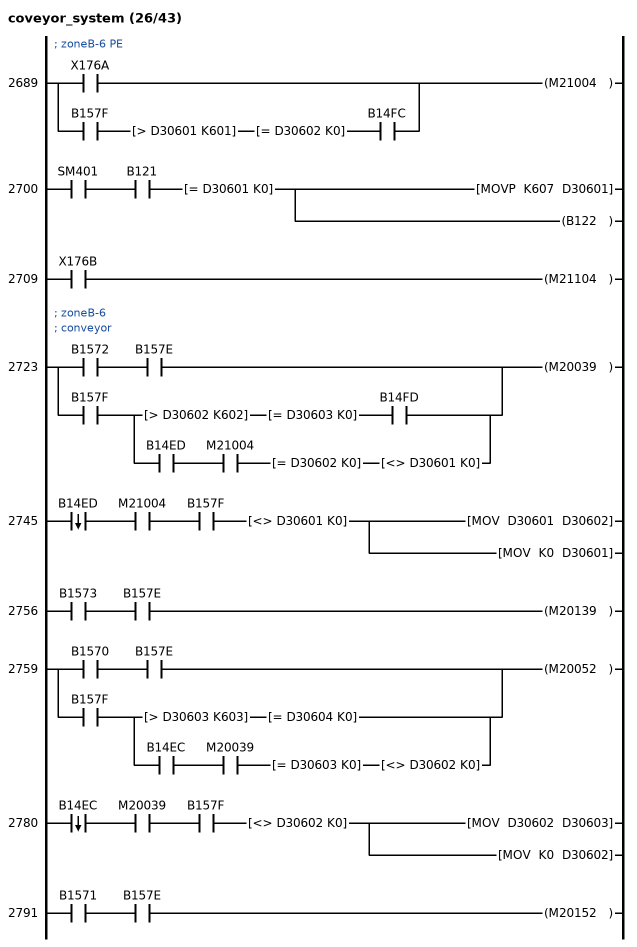
[picture p192: ladder of coveyor_system, rungs at steps 2689 to 2791]
; zoneB-6 PE
2689  LD      X176A
      LD      B157F
      AND>    D30601 K601
      AND=    D30602 K0
      AND     B14FC
      ORB
      OUT     M21004
2700  LD      SM401
      AND     B121
      AND=    D30601 K0
      MOVP    K607 D30601
      OUT     B122
2709  LD      X176B
      OUT     M21104
; zoneB-6
; conveyor
2723  LD      B1572
      AND     B157E
      LD      B157F
      LD>     D30602 K602
      AND=    D30603 K0
      AND     B14FD
      LD      B14ED
      AND     M21004
      AND=    D30602 K0
      AND<>   D30601 K0
      ORB
      ANB
      ORB
      OUT     M20039
2745  LDF     B14ED
      AND     M21004
      AND     B157F
      AND<>   D30601 K0
      MOV     D30601 D30602
      MOV     K0 D30601
2756  LD      B1573
      AND     B157E
      OUT     M20139
2759  LD      B1570
      AND     B157E
      LD      B157F
      LD>     D30603 K603
      AND=    D30604 K0
      LD      B14EC
      AND     M20039
      AND=    D30603 K0
      AND<>   D30602 K0
      ORB
      ANB
      ORB
      OUT     M20052
2780  LDF     B14EC
      AND     M20039
      AND     B157F
      AND<>   D30602 K0
      MOV     D30602 D30603
      MOV     K0 D30602
2791  LD      B1571
      AND     B157E
      OUT     M20152
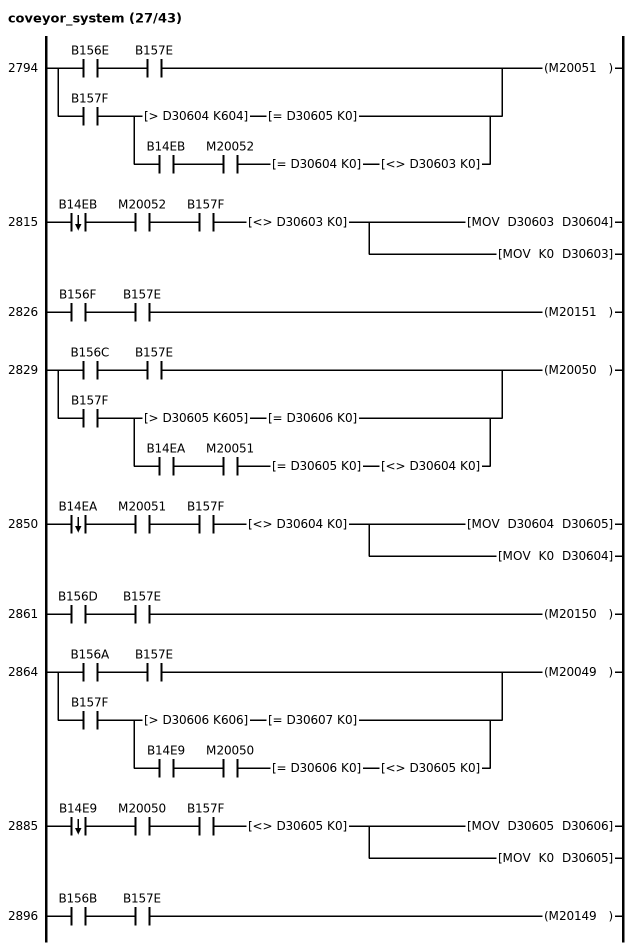
2794  LD      B156E
      AND     B157E
      LD      B157F
      LD>     D30604 K604
      AND=    D30605 K0
      LD      B14EB
      AND     M20052
      AND=    D30604 K0
      AND<>   D30603 K0
      ORB
      ANB
      ORB
      OUT     M20051
2815  LDF     B14EB
      AND     M20052
      AND     B157F
      AND<>   D30603 K0
      MOV     D30603 D30604
      MOV     K0 D30603
2826  LD      B156F
      AND     B157E
      OUT     M20151
2829  LD      B156C
      AND     B157E
      LD      B157F
      LD>     D30605 K605
      AND=    D30606 K0
      LD      B14EA
      AND     M20051
      AND=    D30605 K0
      AND<>   D30604 K0
      ORB
      ANB
      ORB
      OUT     M20050
2850  LDF     B14EA
      AND     M20051
      AND     B157F
      AND<>   D30604 K0
      MOV     D30604 D30605
      MOV     K0 D30604
2861  LD      B156D
      AND     B157E
      OUT     M20150
2864  LD      B156A
      AND     B157E
      LD      B157F
      LD>     D30606 K606
      AND=    D30607 K0
      LD      B14E9
      AND     M20050
      AND=    D30606 K0
      AND<>   D30605 K0
      ORB
      ANB
      ORB
      OUT     M20049
2885  LDF     B14E9
      AND     M20050
      AND     B157F
      AND<>   D30605 K0
      MOV     D30605 D30606
      MOV     K0 D30605
2896  LD      B156B
      AND     B157E
      OUT     M20149
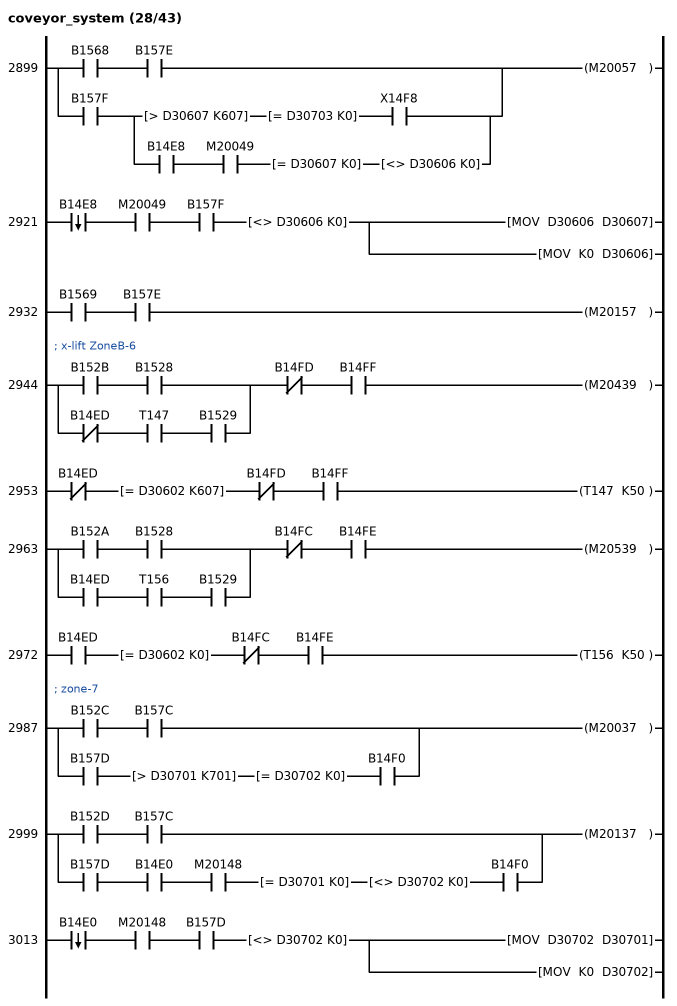
2899  LD      B1568
      AND     B157E
      LD      B157F
      LD>     D30607 K607
      AND=    D30703 K0
      AND     X14F8
      LD      B14E8
      AND     M20049
      AND=    D30607 K0
      AND<>   D30606 K0
      ORB
      ANB
      ORB
      OUT     M20057
2921  LDF     B14E8
      AND     M20049
      AND     B157F
      AND<>   D30606 K0
      MOV     D30606 D30607
      MOV     K0 D30606
2932  LD      B1569
      AND     B157E
      OUT     M20157
; x-lift ZoneB-6
2944  LD      B152B
      AND     B1528
      LDI     B14ED
      AND     T147
      AND     B1529
      ORB
      ANI     B14FD
      AND     B14FF
      OUT     M20439
2953  LDI     B14ED
      AND=    D30602 K607
      ANI     B14FD
      AND     B14FF
      OUT     T147 K50
2963  LD      B152A
      AND     B1528
      LD      B14ED
      AND     T156
      AND     B1529
      ORB
      ANI     B14FC
      AND     B14FE
      OUT     M20539
2972  LD      B14ED
      AND=    D30602 K0
      ANI     B14FC
      AND     B14FE
      OUT     T156 K50
; zone-7
2987  LD      B152C
      AND     B157C
      LD      B157D
      AND>    D30701 K701
      AND=    D30702 K0
      AND     B14F0
      ORB
      OUT     M20037
2999  LD      B152D
      AND     B157C
      LD      B157D
      AND     B14E0
      AND     M20148
      AND=    D30701 K0
      AND<>   D30702 K0
      AND     B14F0
      ORB
      OUT     M20137
3013  LDF     B14E0
      AND     M20148
      AND     B157D
      AND<>   D30702 K0
      MOV     D30702 D30701
      MOV     K0 D30702
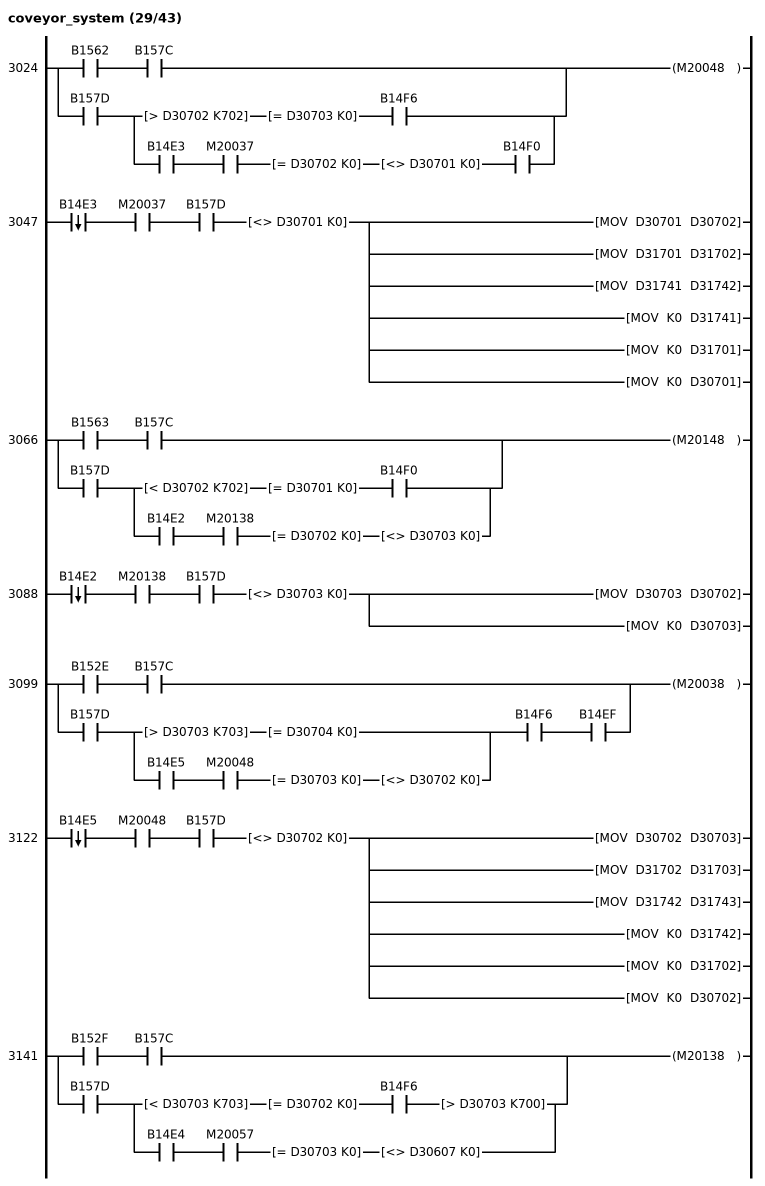
3024  LD      B1562
      AND     B157C
      LD      B157D
      LD>     D30702 K702
      AND=    D30703 K0
      AND     B14F6
      LD      B14E3
      AND     M20037
      AND=    D30702 K0
      AND<>   D30701 K0
      AND     B14F0
      ORB
      ANB
      ORB
      OUT     M20048
3047  LDF     B14E3
      AND     M20037
      AND     B157D
      AND<>   D30701 K0
      MOV     D30701 D30702
      MOV     D31701 D31702
      MOV     D31741 D31742
      MOV     K0 D31741
      MOV     K0 D31701
      MOV     K0 D30701
3066  LD      B1563
      AND     B157C
      LD      B157D
      LD<     D30702 K702
      AND=    D30701 K0
      AND     B14F0
      LD      B14E2
      AND     M20138
      AND=    D30702 K0
      AND<>   D30703 K0
      ORB
      ANB
      ORB
      OUT     M20148
3088  LDF     B14E2
      AND     M20138
      AND     B157D
      AND<>   D30703 K0
      MOV     D30703 D30702
      MOV     K0 D30703
3099  LD      B152E
      AND     B157C
      LD      B157D
      LD>     D30703 K703
      AND=    D30704 K0
      LD      B14E5
      AND     M20048
      AND=    D30703 K0
      AND<>   D30702 K0
      ORB
      ANB
      AND     B14F6
      AND     B14EF
      ORB
      OUT     M20038
3122  LDF     B14E5
      AND     M20048
      AND     B157D
      AND<>   D30702 K0
      MOV     D30702 D30703
      MOV     D31702 D31703
      MOV     D31742 D31743
      MOV     K0 D31742
      MOV     K0 D31702
      MOV     K0 D30702
3141  LD      B152F
      AND     B157C
      LD      B157D
      LD<     D30703 K703
      AND=    D30702 K0
      AND     B14F6
      AND>    D30703 K700
      LD      B14E4
      AND     M20057
      AND=    D30703 K0
      AND<>   D30607 K0
      ORB
      ANB
      ORB
      OUT     M20138
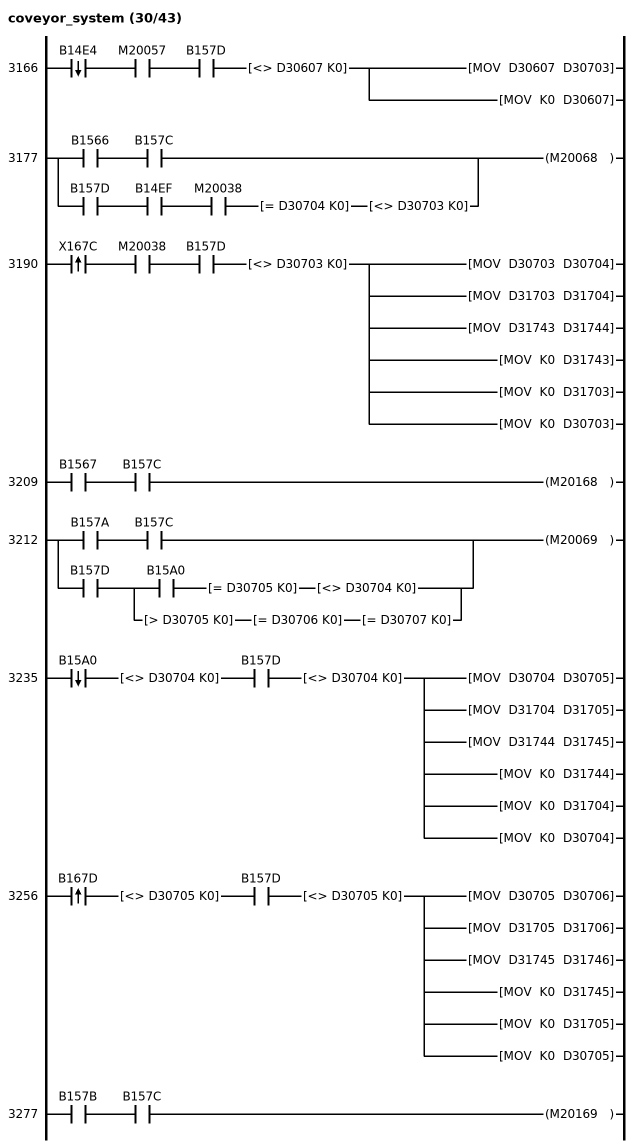
3166  LDF     B14E4
      AND     M20057
      AND     B157D
      AND<>   D30607 K0
      MOV     D30607 D30703
      MOV     K0 D30607
3177  LD      B1566
      AND     B157C
      LD      B157D
      AND     B14EF
      AND     M20038
      AND=    D30704 K0
      AND<>   D30703 K0
      ORB
      OUT     M20068
3190  LDP     X167C
      AND     M20038
      AND     B157D
      AND<>   D30703 K0
      MOV     D30703 D30704
      MOV     D31703 D31704
      MOV     D31743 D31744
      MOV     K0 D31743
      MOV     K0 D31703
      MOV     K0 D30703
3209  LD      B1567
      AND     B157C
      OUT     M20168
3212  LD      B157A
      AND     B157C
      LD      B157D
      LD      B15A0
      AND=    D30705 K0
      AND<>   D30704 K0
      LD>     D30705 K0
      AND=    D30706 K0
      AND=    D30707 K0
      ORB
      ANB
      ORB
      OUT     M20069
3235  LDF     B15A0
      AND<>   D30704 K0
      AND     B157D
      AND<>   D30704 K0
      MOV     D30704 D30705
      MOV     D31704 D31705
      MOV     D31744 D31745
      MOV     K0 D31744
      MOV     K0 D31704
      MOV     K0 D30704
3256  LDP     B167D
      AND<>   D30705 K0
      AND     B157D
      AND<>   D30705 K0
      MOV     D30705 D30706
      MOV     D31705 D31706
      MOV     D31745 D31746
      MOV     K0 D31745
      MOV     K0 D31705
      MOV     K0 D30705
3277  LD      B157B
      AND     B157C
      OUT     M20169
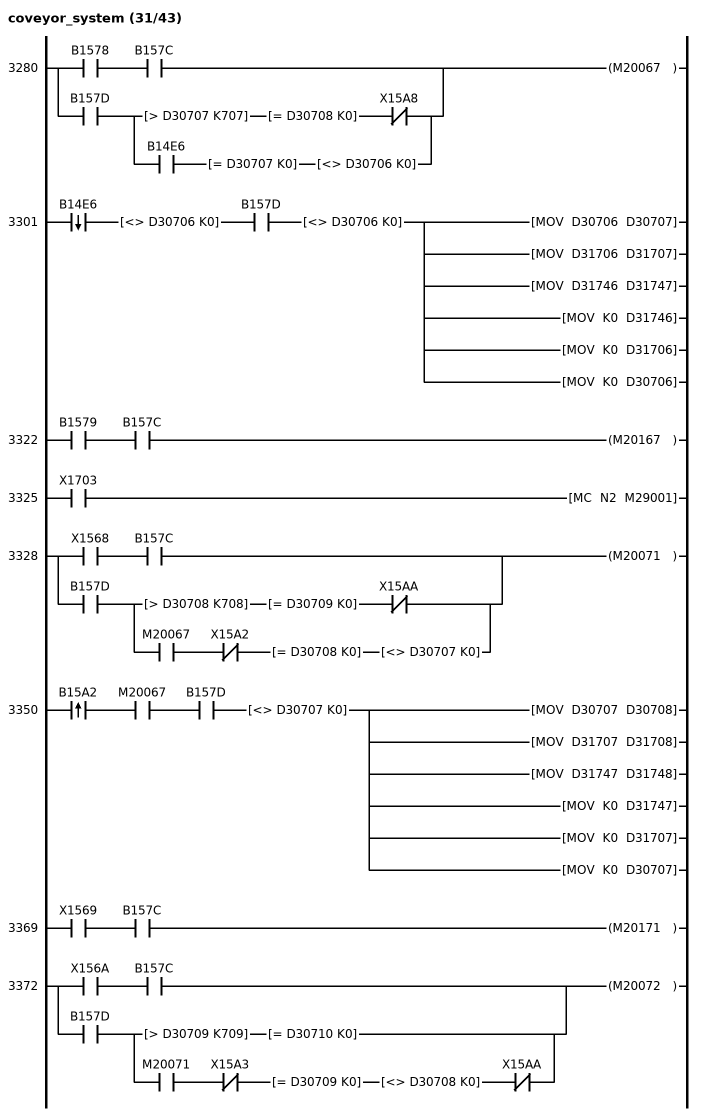
3280  LD      B1578
      AND     B157C
      LD      B157D
      LD>     D30707 K707
      AND=    D30708 K0
      ANI     X15A8
      LD      B14E6
      AND=    D30707 K0
      AND<>   D30706 K0
      ORB
      ANB
      ORB
      OUT     M20067
3301  LDF     B14E6
      AND<>   D30706 K0
      AND     B157D
      AND<>   D30706 K0
      MOV     D30706 D30707
      MOV     D31706 D31707
      MOV     D31746 D31747
      MOV     K0 D31746
      MOV     K0 D31706
      MOV     K0 D30706
3322  LD      B1579
      AND     B157C
      OUT     M20167
3325  LD      X1703
      MC      N2 M29001
3328  LD      X1568
      AND     B157C
      LD      B157D
      LD>     D30708 K708
      AND=    D30709 K0
      ANI     X15AA
      LD      M20067
      ANI     X15A2
      AND=    D30708 K0
      AND<>   D30707 K0
      ORB
      ANB
      ORB
      OUT     M20071
3350  LDP     B15A2
      AND     M20067
      AND     B157D
      AND<>   D30707 K0
      MOV     D30707 D30708
      MOV     D31707 D31708
      MOV     D31747 D31748
      MOV     K0 D31747
      MOV     K0 D31707
      MOV     K0 D30707
3369  LD      X1569
      AND     B157C
      OUT     M20171
3372  LD      X156A
      AND     B157C
      LD      B157D
      LD>     D30709 K709
      AND=    D30710 K0
      LD      M20071
      ANI     X15A3
      AND=    D30709 K0
      AND<>   D30708 K0
      ANI     X15AA
      ORB
      ANB
      ORB
      OUT     M20072
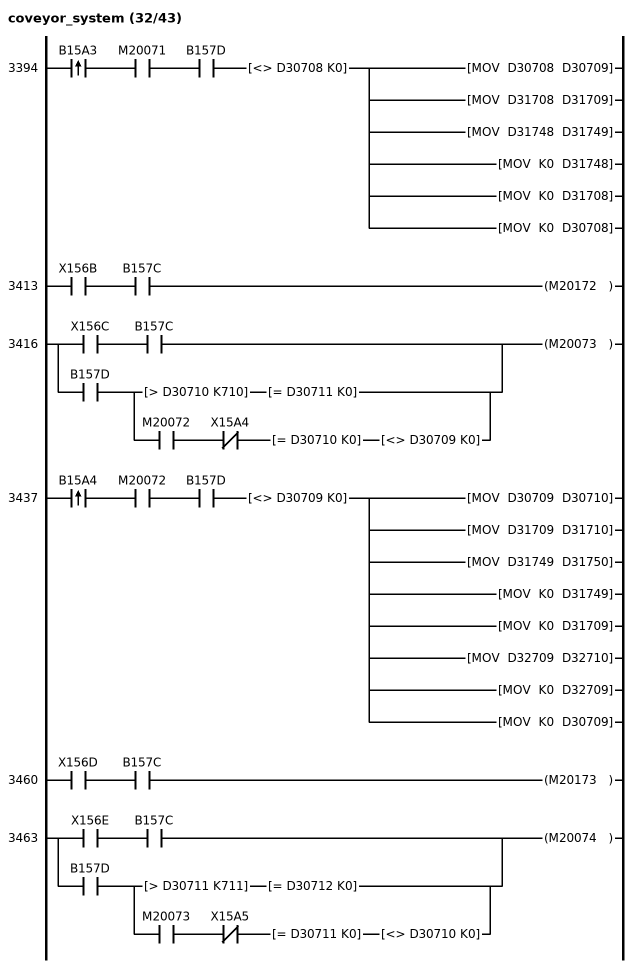
3394  LDP     B15A3
      AND     M20071
      AND     B157D
      AND<>   D30708 K0
      MOV     D30708 D30709
      MOV     D31708 D31709
      MOV     D31748 D31749
      MOV     K0 D31748
      MOV     K0 D31708
      MOV     K0 D30708
3413  LD      X156B
      AND     B157C
      OUT     M20172
3416  LD      X156C
      AND     B157C
      LD      B157D
      LD>     D30710 K710
      AND=    D30711 K0
      LD      M20072
      ANI     X15A4
      AND=    D30710 K0
      AND<>   D30709 K0
      ORB
      ANB
      ORB
      OUT     M20073
3437  LDP     B15A4
      AND     M20072
      AND     B157D
      AND<>   D30709 K0
      MOV     D30709 D30710
      MOV     D31709 D31710
      MOV     D31749 D31750
      MOV     K0 D31749
      MOV     K0 D31709
      MOV     D32709 D32710
      MOV     K0 D32709
      MOV     K0 D30709
3460  LD      X156D
      AND     B157C
      OUT     M20173
3463  LD      X156E
      AND     B157C
      LD      B157D
      LD>     D30711 K711
      AND=    D30712 K0
      LD      M20073
      ANI     X15A5
      AND=    D30711 K0
      AND<>   D30710 K0
      ORB
      ANB
      ORB
      OUT     M20074
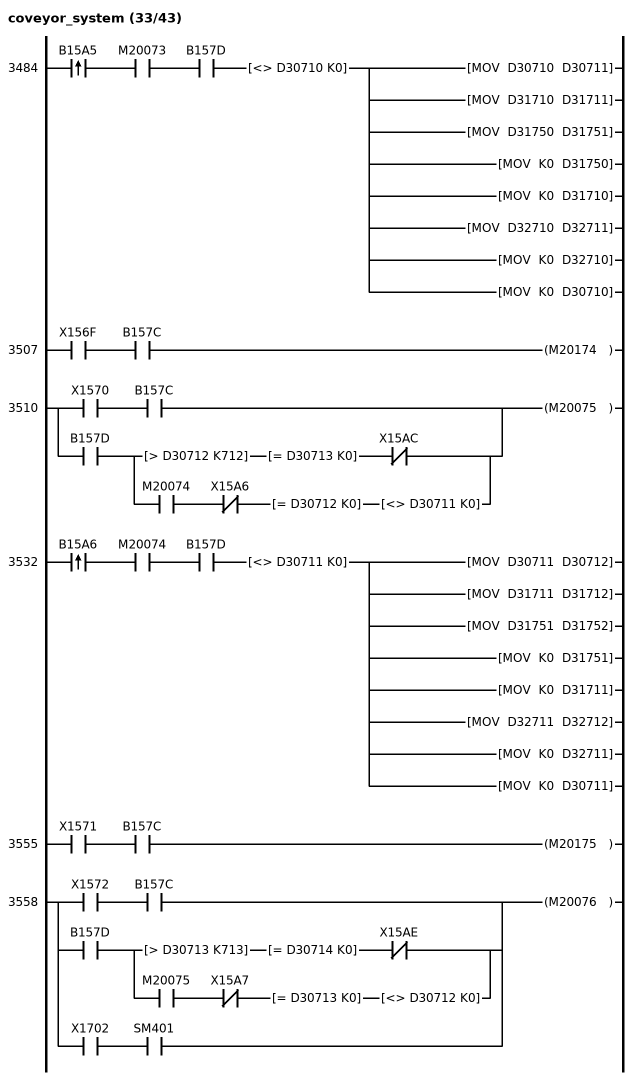
3484  LDP     B15A5
      AND     M20073
      AND     B157D
      AND<>   D30710 K0
      MOV     D30710 D30711
      MOV     D31710 D31711
      MOV     D31750 D31751
      MOV     K0 D31750
      MOV     K0 D31710
      MOV     D32710 D32711
      MOV     K0 D32710
      MOV     K0 D30710
3507  LD      X156F
      AND     B157C
      OUT     M20174
3510  LD      X1570
      AND     B157C
      LD      B157D
      LD>     D30712 K712
      AND=    D30713 K0
      ANI     X15AC
      LD      M20074
      ANI     X15A6
      AND=    D30712 K0
      AND<>   D30711 K0
      ORB
      ANB
      ORB
      OUT     M20075
3532  LDP     B15A6
      AND     M20074
      AND     B157D
      AND<>   D30711 K0
      MOV     D30711 D30712
      MOV     D31711 D31712
      MOV     D31751 D31752
      MOV     K0 D31751
      MOV     K0 D31711
      MOV     D32711 D32712
      MOV     K0 D32711
      MOV     K0 D30711
3555  LD      X1571
      AND     B157C
      OUT     M20175
3558  LD      X1572
      AND     B157C
      LD      B157D
      LD>     D30713 K713
      AND=    D30714 K0
      ANI     X15AE
      LD      M20075
      ANI     X15A7
      AND=    D30713 K0
      AND<>   D30712 K0
      ORB
      ANB
      ORB
      LD      X1702
      AND     SM401
      ORB
      OUT     M20076
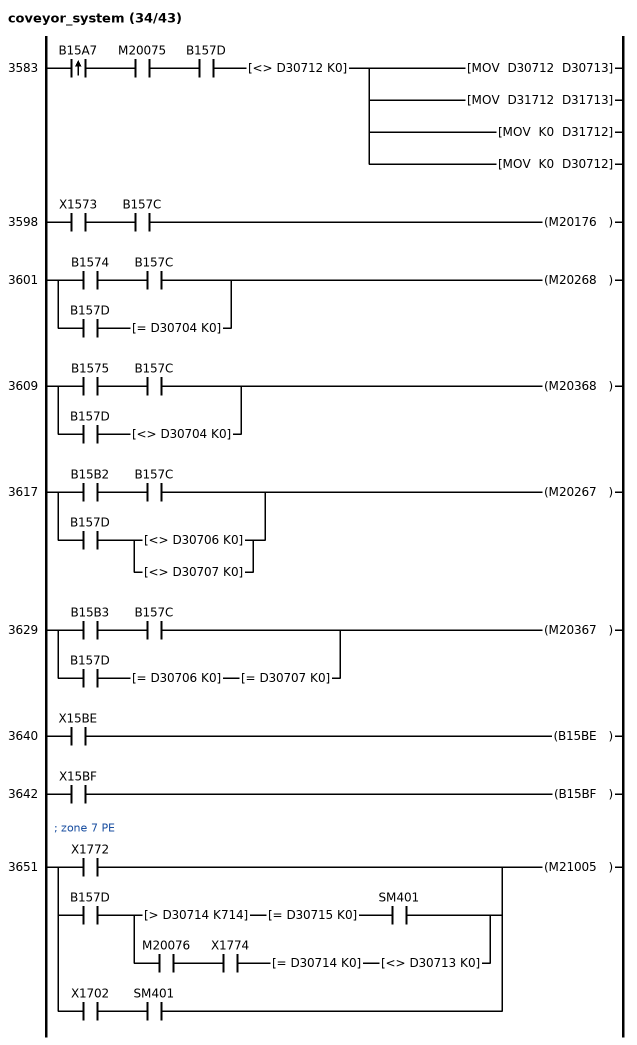
3583  LDP     B15A7
      AND     M20075
      AND     B157D
      AND<>   D30712 K0
      MOV     D30712 D30713
      MOV     D31712 D31713
      MOV     K0 D31712
      MOV     K0 D30712
3598  LD      X1573
      AND     B157C
      OUT     M20176
3601  LD      B1574
      AND     B157C
      LD      B157D
      AND=    D30704 K0
      ORB
      OUT     M20268
3609  LD      B1575
      AND     B157C
      LD      B157D
      AND<>   D30704 K0
      ORB
      OUT     M20368
3617  LD      B15B2
      AND     B157C
      LD      B157D
      LD<>    D30706 K0
      OR<>    D30707 K0
      ANB
      ORB
      OUT     M20267
3629  LD      B15B3
      AND     B157C
      LD      B157D
      AND=    D30706 K0
      AND=    D30707 K0
      ORB
      OUT     M20367
3640  LD      X15BE
      OUT     B15BE
3642  LD      X15BF
      OUT     B15BF
; zone 7 PE
3651  LD      X1772
      LD      B157D
      LD>     D30714 K714
      AND=    D30715 K0
      AND     SM401
      LD      M20076
      AND     X1774
      AND=    D30714 K0
      AND<>   D30713 K0
      ORB
      ANB
      ORB
      LD      X1702
      AND     SM401
      ORB
      OUT     M21005
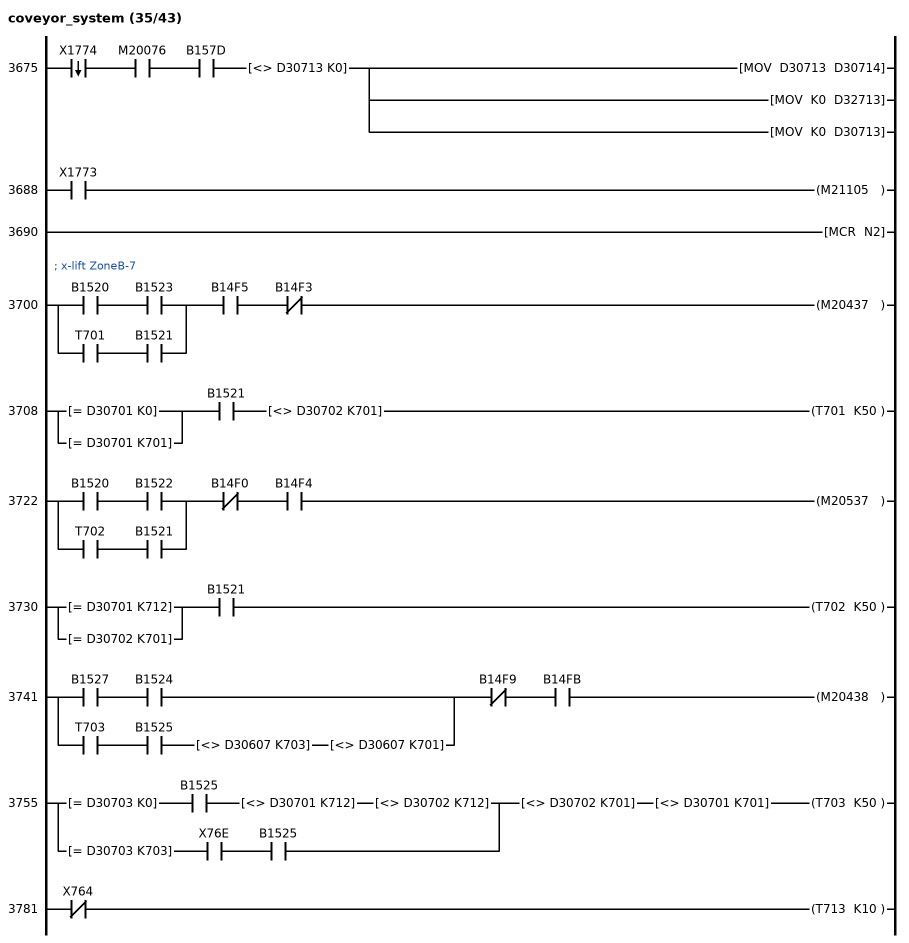
3675  LDF     X1774
      AND     M20076
      AND     B157D
      AND<>   D30713 K0
      MOV     D30713 D30714
      MOV     K0 D32713
      MOV     K0 D30713
3688  LD      X1773
      OUT     M21105
3690  MCR     N2
; x-lift ZoneB-7
3700  LD      B1520
      AND     B1523
      LD      T701
      AND     B1521
      ORB
      AND     B14F5
      ANI     B14F3
      OUT     M20437
3708  LD=     D30701 K0
      OR=     D30701 K701
      AND     B1521
      AND<>   D30702 K701
      OUT     T701 K50
3722  LD      B1520
      AND     B1522
      LD      T702
      AND     B1521
      ORB
      ANI     B14F0
      AND     B14F4
      OUT     M20537
3730  LD=     D30701 K712
      OR=     D30702 K701
      AND     B1521
      OUT     T702 K50
3741  LD      B1527
      AND     B1524
      LD      T703
      AND     B1525
      AND<>   D30607 K703
      AND<>   D30607 K701
      ORB
      ANI     B14F9
      AND     B14FB
      OUT     M20438
3755  LD=     D30703 K0
      AND     B1525
      AND<>   D30701 K712
      AND<>   D30702 K712
      LD=     D30703 K703
      AND     X76E
      AND     B1525
      ORB
      AND<>   D30702 K701
      AND<>   D30701 K701
      OUT     T703 K50
3781  LDI     X764
      OUT     T713 K10
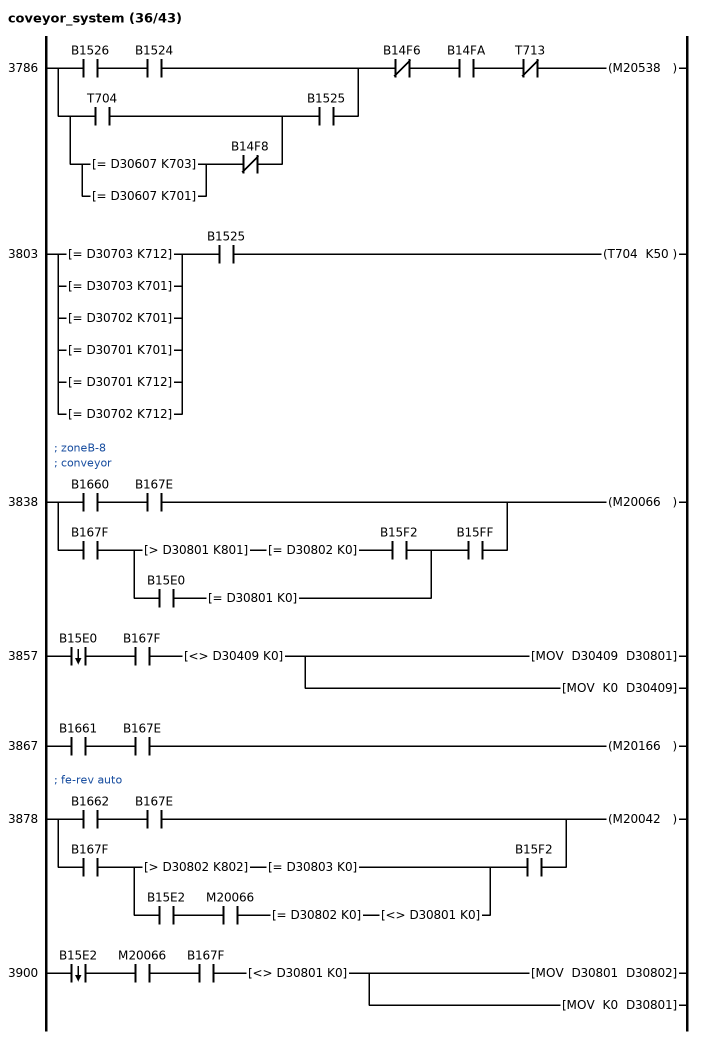
3786  LD      B1526
      AND     B1524
      LD      T704
      LD=     D30607 K703
      OR=     D30607 K701
      ANI     B14F8
      ORB
      AND     B1525
      ORB
      ANI     B14F6
      AND     B14FA
      ANI     T713
      OUT     M20538
3803  LD=     D30703 K712
      OR=     D30703 K701
      OR=     D30702 K701
      OR=     D30701 K701
      OR=     D30701 K712
      OR=     D30702 K712
      AND     B1525
      OUT     T704 K50
; zoneB-8
; conveyor
3838  LD      B1660
      AND     B167E
      LD      B167F
      LD>     D30801 K801
      AND=    D30802 K0
      AND     B15F2
      LD      B15E0
      AND=    D30801 K0
      ORB
      ANB
      AND     B15FF
      ORB
      OUT     M20066
3857  LDF     B15E0
      AND     B167F
      AND<>   D30409 K0
      MOV     D30409 D30801
      MOV     K0 D30409
3867  LD      B1661
      AND     B167E
      OUT     M20166
; fe-rev auto
3878  LD      B1662
      AND     B167E
      LD      B167F
      LD>     D30802 K802
      AND=    D30803 K0
      LD      B15E2
      AND     M20066
      AND=    D30802 K0
      AND<>   D30801 K0
      ORB
      ANB
      AND     B15F2
      ORB
      OUT     M20042
3900  LDF     B15E2
      AND     M20066
      AND     B167F
      AND<>   D30801 K0
      MOV     D30801 D30802
      MOV     K0 D30801
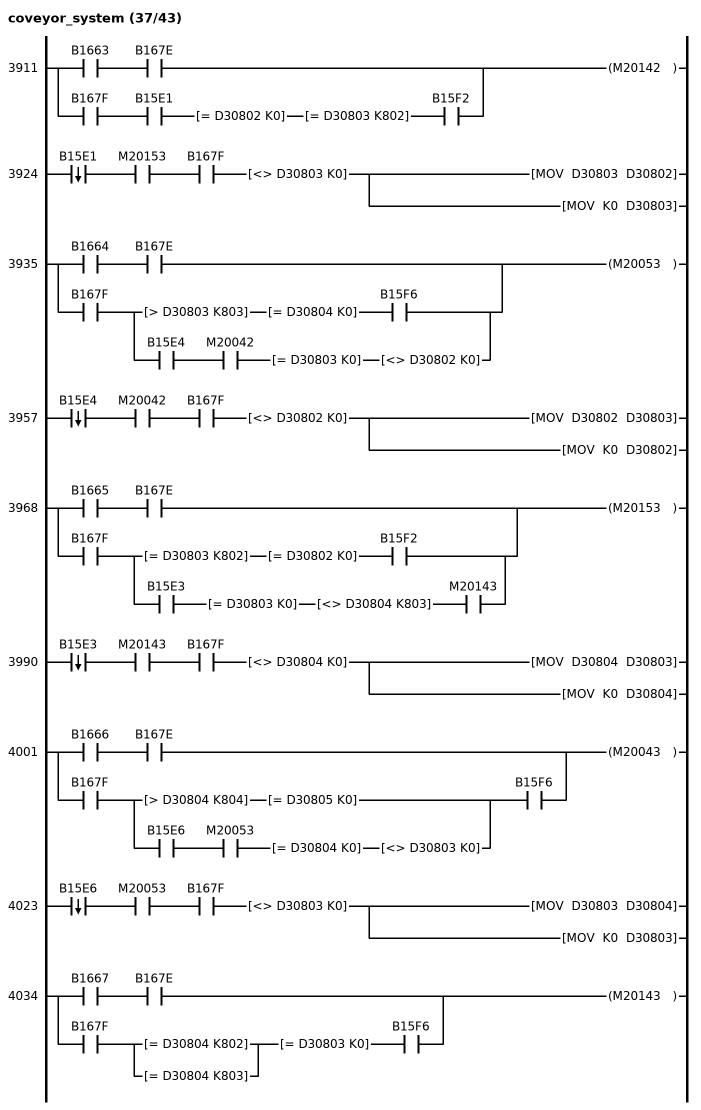
3911  LD      B1663
      AND     B167E
      LD      B167F
      AND     B15E1
      AND=    D30802 K0
      AND=    D30803 K802
      AND     B15F2
      ORB
      OUT     M20142
3924  LDF     B15E1
      AND     M20153
      AND     B167F
      AND<>   D30803 K0
      MOV     D30803 D30802
      MOV     K0 D30803
3935  LD      B1664
      AND     B167E
      LD      B167F
      LD>     D30803 K803
      AND=    D30804 K0
      AND     B15F6
      LD      B15E4
      AND     M20042
      AND=    D30803 K0
      AND<>   D30802 K0
      ORB
      ANB
      ORB
      OUT     M20053
3957  LDF     B15E4
      AND     M20042
      AND     B167F
      AND<>   D30802 K0
      MOV     D30802 D30803
      MOV     K0 D30802
3968  LD      B1665
      AND     B167E
      LD      B167F
      LD=     D30803 K802
      AND=    D30802 K0
      AND     B15F2
      LD      B15E3
      AND=    D30803 K0
      AND<>   D30804 K803
      AND     M20143
      ORB
      ANB
      ORB
      OUT     M20153
3990  LDF     B15E3
      AND     M20143
      AND     B167F
      AND<>   D30804 K0
      MOV     D30804 D30803
      MOV     K0 D30804
4001  LD      B1666
      AND     B167E
      LD      B167F
      LD>     D30804 K804
      AND=    D30805 K0
      LD      B15E6
      AND     M20053
      AND=    D30804 K0
      AND<>   D30803 K0
      ORB
      ANB
      AND     B15F6
      ORB
      OUT     M20043
4023  LDF     B15E6
      AND     M20053
      AND     B167F
      AND<>   D30803 K0
      MOV     D30803 D30804
      MOV     K0 D30803
4034  LD      B1667
      AND     B167E
      LD      B167F
      LD=     D30804 K802
      OR=     D30804 K803
      ANB
      AND=    D30803 K0
      AND     B15F6
      ORB
      OUT     M20143
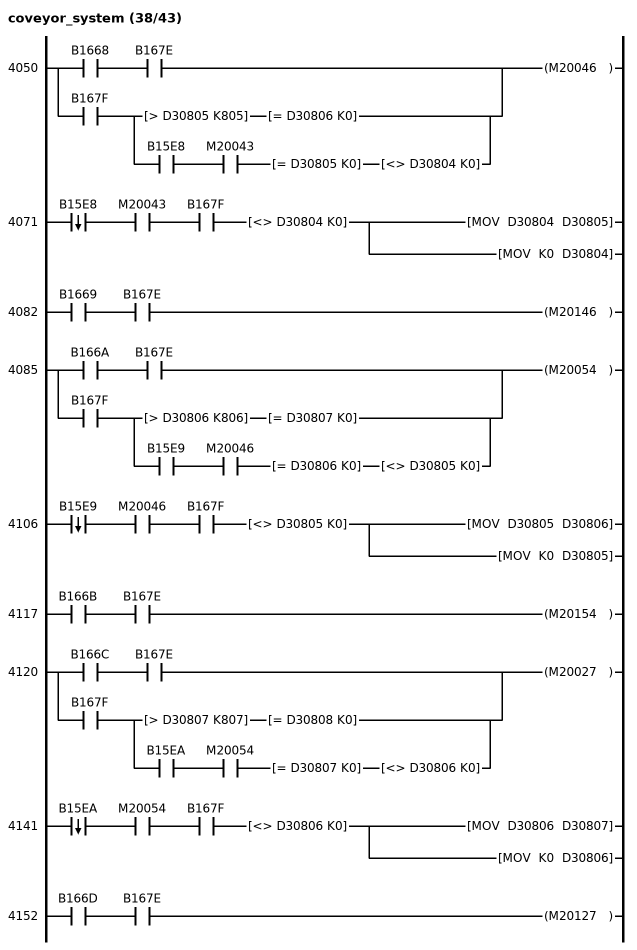
4050  LD      B1668
      AND     B167E
      LD      B167F
      LD>     D30805 K805
      AND=    D30806 K0
      LD      B15E8
      AND     M20043
      AND=    D30805 K0
      AND<>   D30804 K0
      ORB
      ANB
      ORB
      OUT     M20046
4071  LDF     B15E8
      AND     M20043
      AND     B167F
      AND<>   D30804 K0
      MOV     D30804 D30805
      MOV     K0 D30804
4082  LD      B1669
      AND     B167E
      OUT     M20146
4085  LD      B166A
      AND     B167E
      LD      B167F
      LD>     D30806 K806
      AND=    D30807 K0
      LD      B15E9
      AND     M20046
      AND=    D30806 K0
      AND<>   D30805 K0
      ORB
      ANB
      ORB
      OUT     M20054
4106  LDF     B15E9
      AND     M20046
      AND     B167F
      AND<>   D30805 K0
      MOV     D30805 D30806
      MOV     K0 D30805
4117  LD      B166B
      AND     B167E
      OUT     M20154
4120  LD      B166C
      AND     B167E
      LD      B167F
      LD>     D30807 K807
      AND=    D30808 K0
      LD      B15EA
      AND     M20054
      AND=    D30807 K0
      AND<>   D30806 K0
      ORB
      ANB
      ORB
      OUT     M20027
4141  LDF     B15EA
      AND     M20054
      AND     B167F
      AND<>   D30806 K0
      MOV     D30806 D30807
      MOV     K0 D30806
4152  LD      B166D
      AND     B167E
      OUT     M20127
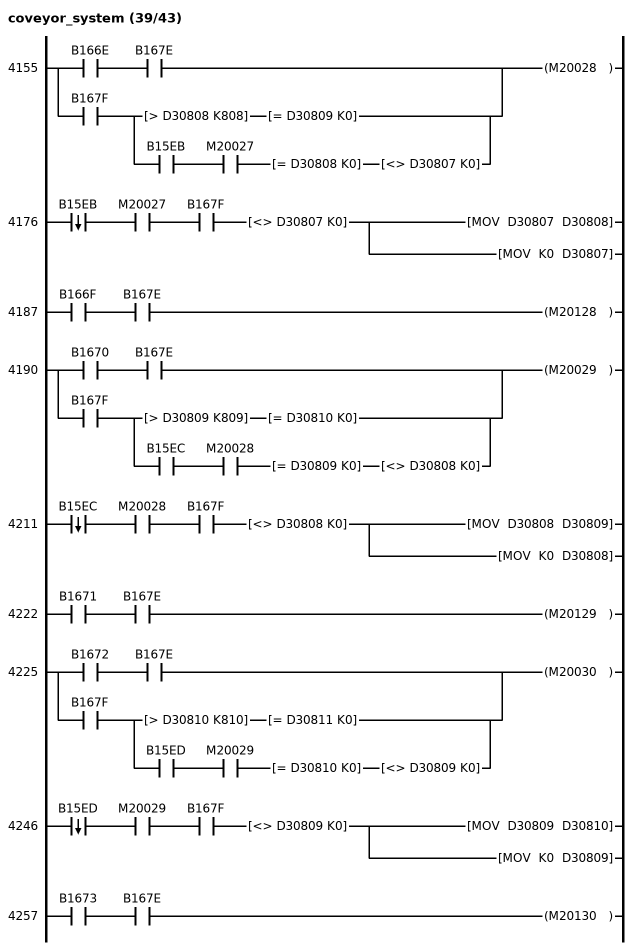
4155  LD      B166E
      AND     B167E
      LD      B167F
      LD>     D30808 K808
      AND=    D30809 K0
      LD      B15EB
      AND     M20027
      AND=    D30808 K0
      AND<>   D30807 K0
      ORB
      ANB
      ORB
      OUT     M20028
4176  LDF     B15EB
      AND     M20027
      AND     B167F
      AND<>   D30807 K0
      MOV     D30807 D30808
      MOV     K0 D30807
4187  LD      B166F
      AND     B167E
      OUT     M20128
4190  LD      B1670
      AND     B167E
      LD      B167F
      LD>     D30809 K809
      AND=    D30810 K0
      LD      B15EC
      AND     M20028
      AND=    D30809 K0
      AND<>   D30808 K0
      ORB
      ANB
      ORB
      OUT     M20029
4211  LDF     B15EC
      AND     M20028
      AND     B167F
      AND<>   D30808 K0
      MOV     D30808 D30809
      MOV     K0 D30808
4222  LD      B1671
      AND     B167E
      OUT     M20129
4225  LD      B1672
      AND     B167E
      LD      B167F
      LD>     D30810 K810
      AND=    D30811 K0
      LD      B15ED
      AND     M20029
      AND=    D30810 K0
      AND<>   D30809 K0
      ORB
      ANB
      ORB
      OUT     M20030
4246  LDF     B15ED
      AND     M20029
      AND     B167F
      AND<>   D30809 K0
      MOV     D30809 D30810
      MOV     K0 D30809
4257  LD      B1673
      AND     B167E
      OUT     M20130
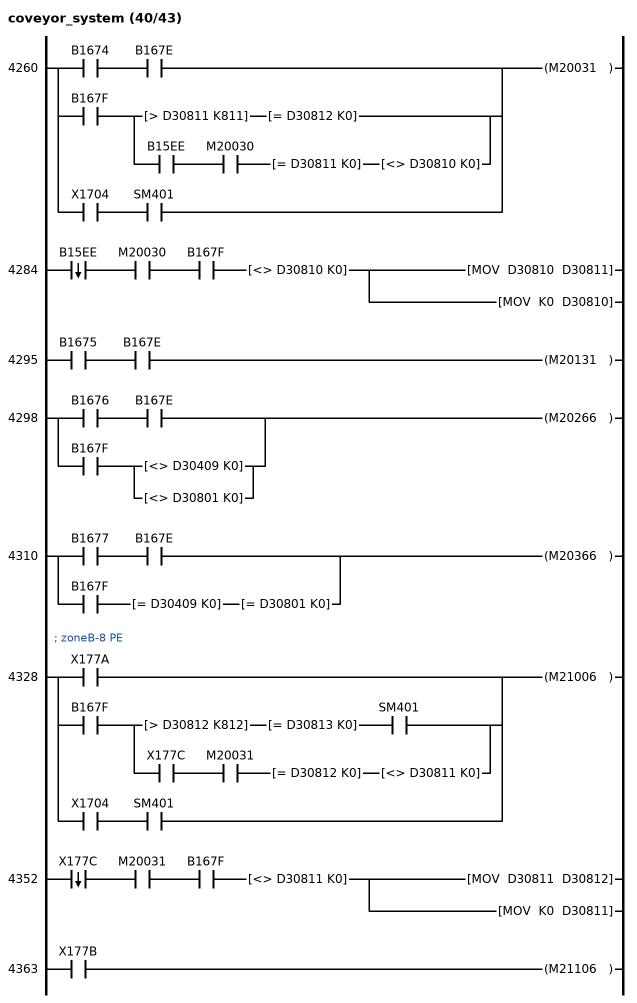
4260  LD      B1674
      AND     B167E
      LD      B167F
      LD>     D30811 K811
      AND=    D30812 K0
      LD      B15EE
      AND     M20030
      AND=    D30811 K0
      AND<>   D30810 K0
      ORB
      ANB
      ORB
      LD      X1704
      AND     SM401
      ORB
      OUT     M20031
4284  LDF     B15EE
      AND     M20030
      AND     B167F
      AND<>   D30810 K0
      MOV     D30810 D30811
      MOV     K0 D30810
4295  LD      B1675
      AND     B167E
      OUT     M20131
4298  LD      B1676
      AND     B167E
      LD      B167F
      LD<>    D30409 K0
      OR<>    D30801 K0
      ANB
      ORB
      OUT     M20266
4310  LD      B1677
      AND     B167E
      LD      B167F
      AND=    D30409 K0
      AND=    D30801 K0
      ORB
      OUT     M20366
; zoneB-8 PE
4328  LD      X177A
      LD      B167F
      LD>     D30812 K812
      AND=    D30813 K0
      AND     SM401
      LD      X177C
      AND     M20031
      AND=    D30812 K0
      AND<>   D30811 K0
      ORB
      ANB
      ORB
      LD      X1704
      AND     SM401
      ORB
      OUT     M21006
4352  LDF     X177C
      AND     M20031
      AND     B167F
      AND<>   D30811 K0
      MOV     D30811 D30812
      MOV     K0 D30811
4363  LD      X177B
      OUT     M21106
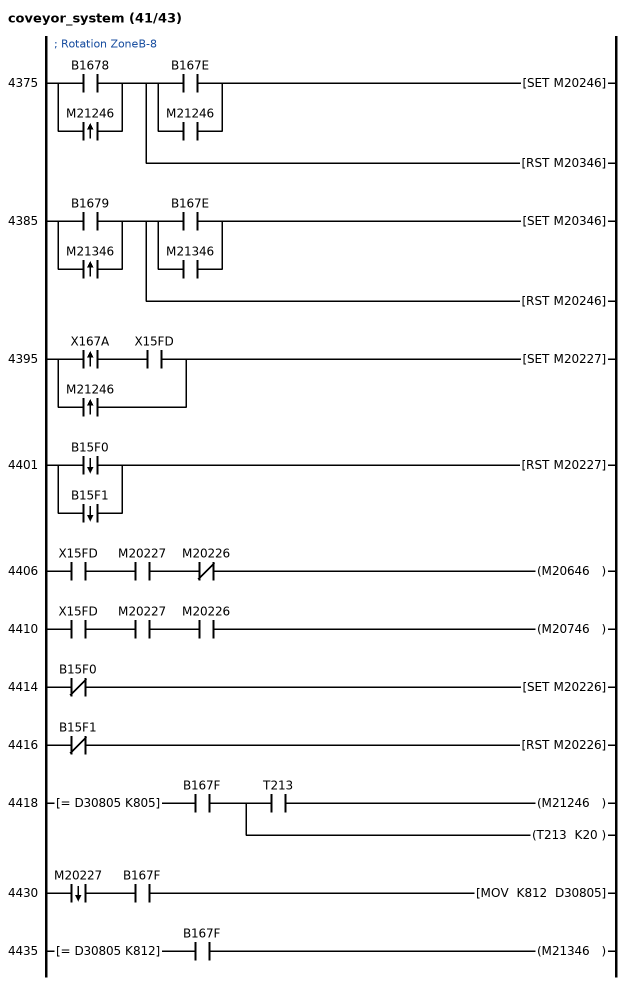
; Rotation ZoneB-8
4375  LD      B1678
      ORP     M21246
      MPS
      LD      B167E
      OR      M21246
      ANB
      SET     M20246
      MPP
      RST     M20346
4385  LD      B1679
      ORP     M21346
      MPS
      LD      B167E
      OR      M21346
      ANB
      SET     M20346
      MPP
      RST     M20246
4395  LDP     X167A
      AND     X15FD
      ORP     M21246
      SET     M20227
4401  LDF     B15F0
      ORF     B15F1
      RST     M20227
4406  LD      X15FD
      AND     M20227
      ANI     M20226
      OUT     M20646
4410  LD      X15FD
      AND     M20227
      AND     M20226
      OUT     M20746
4414  LDI     B15F0
      SET     M20226
4416  LDI     B15F1
      RST     M20226
4418  LD=     D30805 K805
      AND     B167F
      MPS
      AND     T213
      OUT     M21246
      MPP
      OUT     T213 K20
4430  LDF     M20227
      AND     B167F
      MOV     K812 D30805
4435  LD=     D30805 K812
      AND     B167F
      OUT     M21346
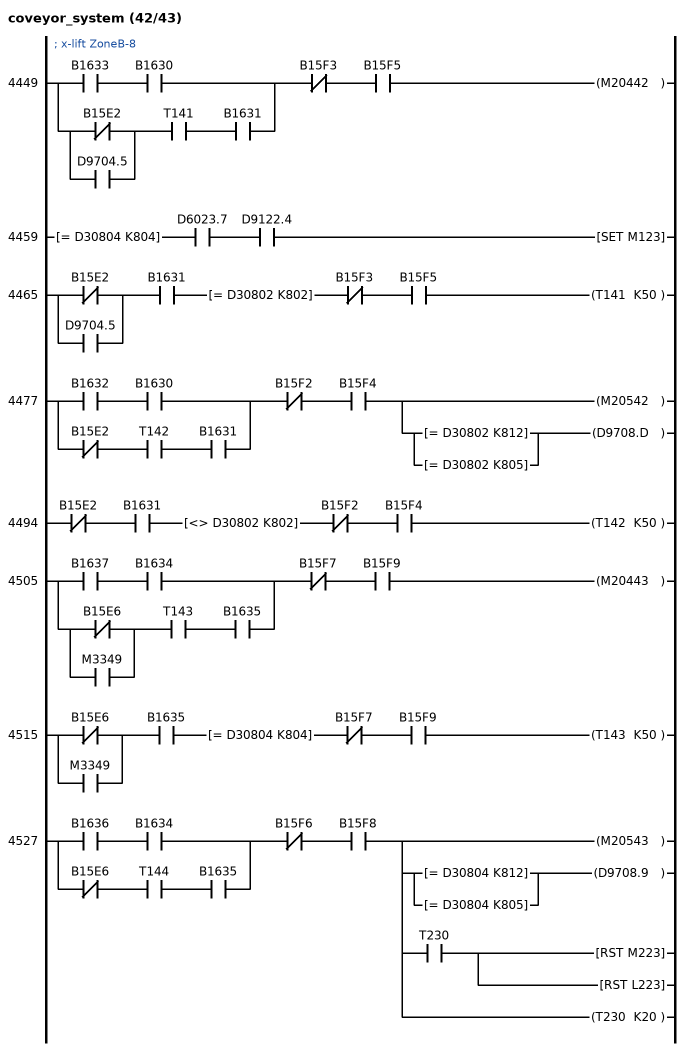
; x-lift ZoneB-8
4449  LD      B1633
      AND     B1630
      LDI     B15E2
      OR      D9704.5
      AND     T141
      AND     B1631
      ORB
      ANI     B15F3
      AND     B15F5
      OUT     M20442
4459  LD=     D30804 K804
      AND     D6023.7
      AND     D9122.4
      SET     M123
4465  LDI     B15E2
      OR      D9704.5
      AND     B1631
      AND=    D30802 K802
      ANI     B15F3
      AND     B15F5
      OUT     T141 K50
4477  LD      B1632
      AND     B1630
      LDI     B15E2
      AND     T142
      AND     B1631
      ORB
      ANI     B15F2
      AND     B15F4
      OUT     M20542
      LD=     D30802 K812
      OR=     D30802 K805
      ANB
      OUT     D9708.D
4494  LDI     B15E2
      AND     B1631
      AND<>   D30802 K802
      ANI     B15F2
      AND     B15F4
      OUT     T142 K50
4505  LD      B1637
      AND     B1634
      LDI     B15E6
      OR      M3349
      AND     T143
      AND     B1635
      ORB
      ANI     B15F7
      AND     B15F9
      OUT     M20443
4515  LDI     B15E6
      OR      M3349
      AND     B1635
      AND=    D30804 K804
      ANI     B15F7
      AND     B15F9
      OUT     T143 K50
4527  LD      B1636
      AND     B1634
      LDI     B15E6
      AND     T144
      AND     B1635
      ORB
      ANI     B15F6
      AND     B15F8
      OUT     M20543
      MPS
      LD=     D30804 K812
      OR=     D30804 K805
      ANB
      OUT     D9708.9
      MRD
      AND     T230
      RST     M223
      RST     L223
      MPP
      OUT     T230 K20
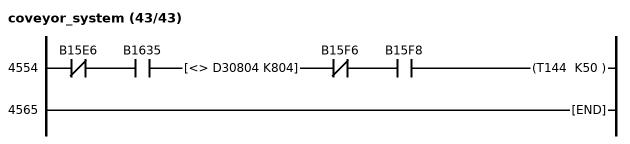
4554  LDI     B15E6
      AND     B1635
      AND<>   D30804 K804
      ANI     B15F6
      AND     B15F8
      OUT     T144 K50
4565  END
END_PROGRAM

PROGRAM data_exchage
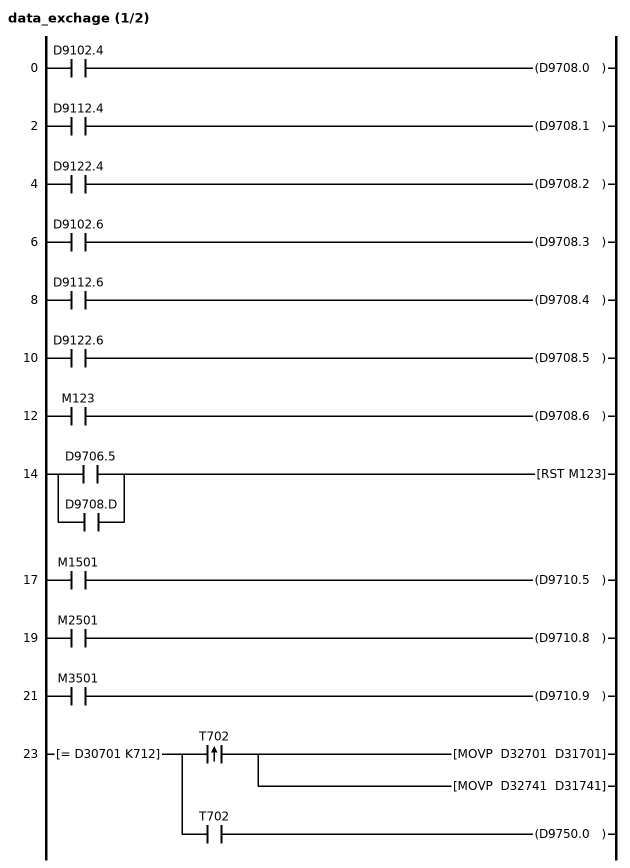
0     LD      D9102.4
      OUT     D9708.0
2     LD      D9112.4
      OUT     D9708.1
4     LD      D9122.4
      OUT     D9708.2
6     LD      D9102.6
      OUT     D9708.3
8     LD      D9112.6
      OUT     D9708.4
10    LD      D9122.6
      OUT     D9708.5
12    LD      M123
      OUT     D9708.6
14    LD      D9706.5
      OR      D9708.D
      RST     M123
17    LD      M1501
      OUT     D9710.5
19    LD      M2501
      OUT     D9710.8
21    LD      M3501
      OUT     D9710.9
23    LD=     D30701 K712
      MPS
      ANDP    T702
      MOVP    D32701 D31701
      MOVP    D32741 D31741
      MPP
      AND     T702
      OUT     D9750.0
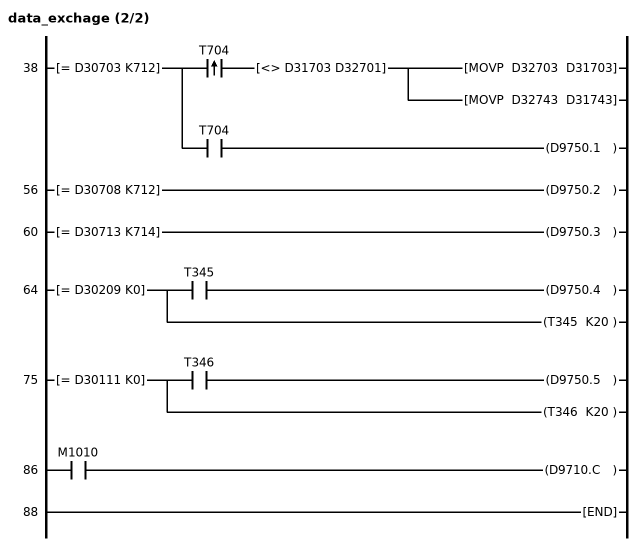
38    LD=     D30703 K712
      MPS
      ANDP    T704
      AND<>   D31703 D32701
      MOVP    D32703 D31703
      MOVP    D32743 D31743
      MPP
      AND     T704
      OUT     D9750.1
56    LD=     D30708 K712
      OUT     D9750.2
60    LD=     D30713 K714
      OUT     D9750.3
64    LD=     D30209 K0
      MPS
      AND     T345
      OUT     D9750.4
      MPP
      OUT     T345 K20
75    LD=     D30111 K0
      MPS
      AND     T346
      OUT     D9750.5
      MPP
      OUT     T346 K20
86    LD      M1010
      OUT     D9710.C
88    END
END_PROGRAM

PROGRAM Display
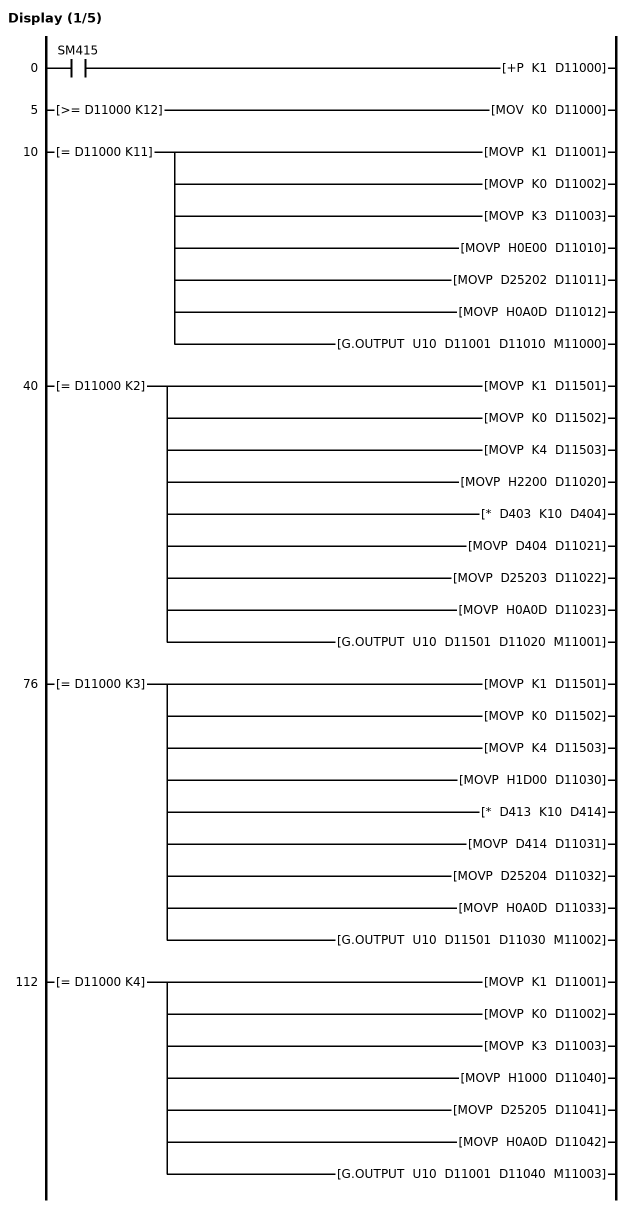
0     LD      SM415
      +P      K1 D11000
5     LD>=    D11000 K12
      MOV     K0 D11000
10    LD=     D11000 K11
      MOVP    K1 D11001
      MOVP    K0 D11002
      MOVP    K3 D11003
      MOVP    H0E00 D11010
      MOVP    D25202 D11011
      MOVP    H0A0D D11012
      G.OUTPUT U10 D11001 D11010 M11000
40    LD=     D11000 K2
      MOVP    K1 D11501
      MOVP    K0 D11502
      MOVP    K4 D11503
      MOVP    H2200 D11020
      *       D403 K10 D404
      MOVP    D404 D11021
      MOVP    D25203 D11022
      MOVP    H0A0D D11023
      G.OUTPUT U10 D11501 D11020 M11001
76    LD=     D11000 K3
      MOVP    K1 D11501
      MOVP    K0 D11502
      MOVP    K4 D11503
      MOVP    H1D00 D11030
      *       D413 K10 D414
      MOVP    D414 D11031
      MOVP    D25204 D11032
      MOVP    H0A0D D11033
      G.OUTPUT U10 D11501 D11030 M11002
112   LD=     D11000 K4
      MOVP    K1 D11001
      MOVP    K0 D11002
      MOVP    K3 D11003
      MOVP    H1000 D11040
      MOVP    D25205 D11041
      MOVP    H0A0D D11042
      G.OUTPUT U10 D11001 D11040 M11003
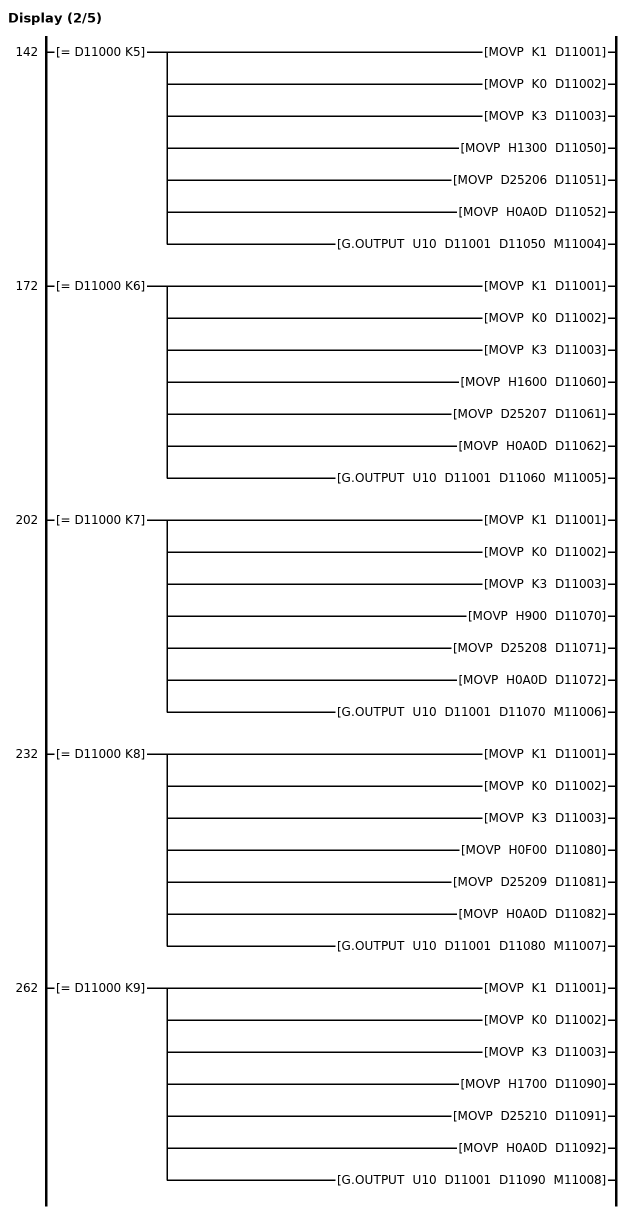
142   LD=     D11000 K5
      MOVP    K1 D11001
      MOVP    K0 D11002
      MOVP    K3 D11003
      MOVP    H1300 D11050
      MOVP    D25206 D11051
      MOVP    H0A0D D11052
      G.OUTPUT U10 D11001 D11050 M11004
172   LD=     D11000 K6
      MOVP    K1 D11001
      MOVP    K0 D11002
      MOVP    K3 D11003
      MOVP    H1600 D11060
      MOVP    D25207 D11061
      MOVP    H0A0D D11062
      G.OUTPUT U10 D11001 D11060 M11005
202   LD=     D11000 K7
      MOVP    K1 D11001
      MOVP    K0 D11002
      MOVP    K3 D11003
      MOVP    H900 D11070
      MOVP    D25208 D11071
      MOVP    H0A0D D11072
      G.OUTPUT U10 D11001 D11070 M11006
232   LD=     D11000 K8
      MOVP    K1 D11001
      MOVP    K0 D11002
      MOVP    K3 D11003
      MOVP    H0F00 D11080
      MOVP    D25209 D11081
      MOVP    H0A0D D11082
      G.OUTPUT U10 D11001 D11080 M11007
262   LD=     D11000 K9
      MOVP    K1 D11001
      MOVP    K0 D11002
      MOVP    K3 D11003
      MOVP    H1700 D11090
      MOVP    D25210 D11091
      MOVP    H0A0D D11092
      G.OUTPUT U10 D11001 D11090 M11008
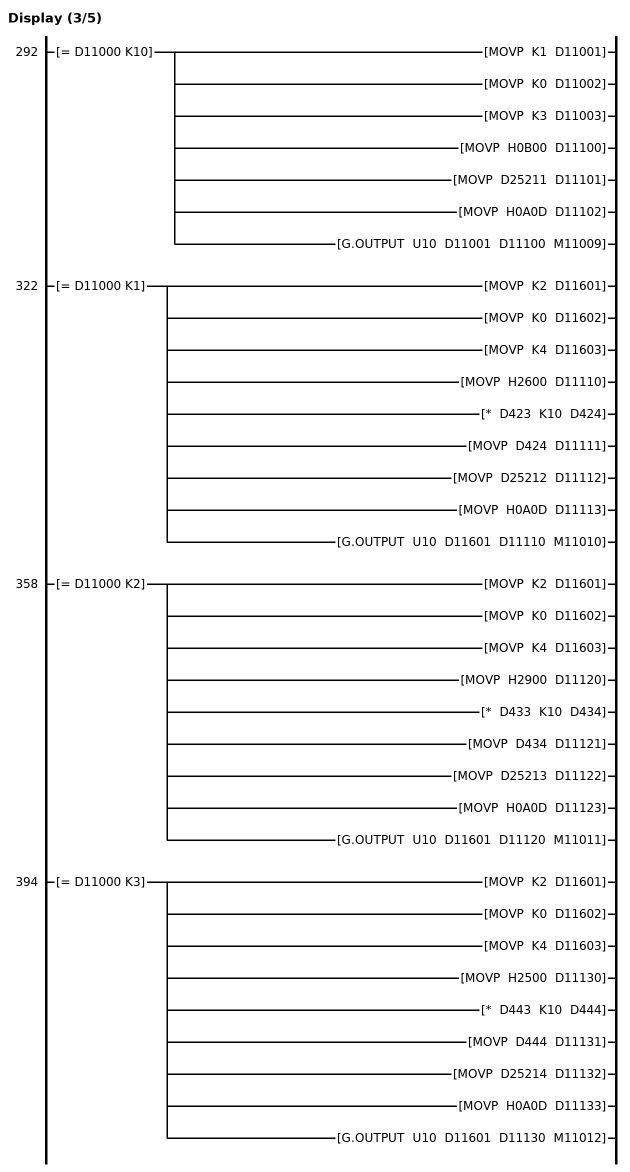
292   LD=     D11000 K10
      MOVP    K1 D11001
      MOVP    K0 D11002
      MOVP    K3 D11003
      MOVP    H0B00 D11100
      MOVP    D25211 D11101
      MOVP    H0A0D D11102
      G.OUTPUT U10 D11001 D11100 M11009
322   LD=     D11000 K1
      MOVP    K2 D11601
      MOVP    K0 D11602
      MOVP    K4 D11603
      MOVP    H2600 D11110
      *       D423 K10 D424
      MOVP    D424 D11111
      MOVP    D25212 D11112
      MOVP    H0A0D D11113
      G.OUTPUT U10 D11601 D11110 M11010
358   LD=     D11000 K2
      MOVP    K2 D11601
      MOVP    K0 D11602
      MOVP    K4 D11603
      MOVP    H2900 D11120
      *       D433 K10 D434
      MOVP    D434 D11121
      MOVP    D25213 D11122
      MOVP    H0A0D D11123
      G.OUTPUT U10 D11601 D11120 M11011
394   LD=     D11000 K3
      MOVP    K2 D11601
      MOVP    K0 D11602
      MOVP    K4 D11603
      MOVP    H2500 D11130
      *       D443 K10 D444
      MOVP    D444 D11131
      MOVP    D25214 D11132
      MOVP    H0A0D D11133
      G.OUTPUT U10 D11601 D11130 M11012
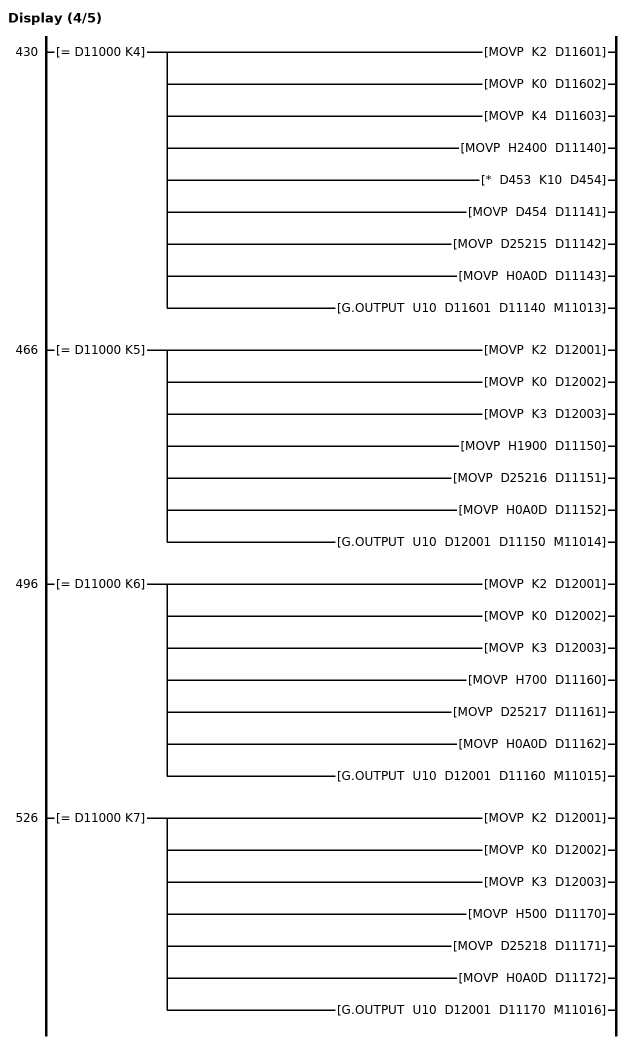
430   LD=     D11000 K4
      MOVP    K2 D11601
      MOVP    K0 D11602
      MOVP    K4 D11603
      MOVP    H2400 D11140
      *       D453 K10 D454
      MOVP    D454 D11141
      MOVP    D25215 D11142
      MOVP    H0A0D D11143
      G.OUTPUT U10 D11601 D11140 M11013
466   LD=     D11000 K5
      MOVP    K2 D12001
      MOVP    K0 D12002
      MOVP    K3 D12003
      MOVP    H1900 D11150
      MOVP    D25216 D11151
      MOVP    H0A0D D11152
      G.OUTPUT U10 D12001 D11150 M11014
496   LD=     D11000 K6
      MOVP    K2 D12001
      MOVP    K0 D12002
      MOVP    K3 D12003
      MOVP    H700 D11160
      MOVP    D25217 D11161
      MOVP    H0A0D D11162
      G.OUTPUT U10 D12001 D11160 M11015
526   LD=     D11000 K7
      MOVP    K2 D12001
      MOVP    K0 D12002
      MOVP    K3 D12003
      MOVP    H500 D11170
      MOVP    D25218 D11171
      MOVP    H0A0D D11172
      G.OUTPUT U10 D12001 D11170 M11016
